PROGRAM MAIN
VAR
	// *** Axis ***
	AxisControl_1: fbAxisControl;

END_VAR

DataProcess();

// *** Axis ***
IF IO.Axis_1.SetVelo = 0 THEN IO.Axis_1.SetVelo := 0.1; END_IF;
AxisControl_1(Axis := IO.Axis_1);

END_PROGRAM

(* stored: Version 1.1.0.1, ProductVersion 3.1.4020.12
   POU MAIN: Id {f41ae2df-d533-4825-87e5-b74800d6223a}, SpecialFunc None *)
